(* Schneider Machine Expert - Basic project P1_Part1C, file version 1.6.0.0 *)
(* ProjectInformations: Name=New project *)

HARDWARE
  Cpu 0: TM221M16R/G
  EthernetConfiguration: NetworkName=M221, IpAllocationMode=FixedAddress, IpAddress=0.0.0.0, SubnetMask=0.0.0.0
  SerialLineConfiguration: Baud=Baud19200, Parity=ParityEven, DataBits=DataBits8, StopBits=StopBits1, PhysicalMedium=PhysicalMediumRs485, TransmissionMode=TransmissionModeModbusRtu, SlaveId=1, Addressing=SlaveAddressing
  MastTask: UsePeriodScanMode=false, PeriodScan=100
  FastTask: Period=255, FastTaskSubroutine=On-Off Loop Timer Control
  CpuBehavior: StartingMode=StartAsPreviousState, AutoSaveRamOnEeprom=true, WatchdogPeriod=250

SYMBOLS  (address, symbol, comment, settings)
  %M0       OUTPUT_0_ST
  %M1       START_TIMER_ON
  %M2       DELAY_TIMER_ON
  %MW0      CURRENT_PRESSURE
  %KW0      PRESSURE_CHECKPOINT  [Value=500]
  %KW1      PRESSURE_CHECKPOINT_UNREACHABLE  [Value=1001]
  %TM0      START_TIMER  [Preset=0, Base=OneSecond]
  %TM1      DELAY_TIMER  [Preset=0, Base=OneSecond]
  %I0.0     INPUT_0
  %Q0.0     OUTPUT_0
  %IW0.0    ON_TIMER  [Type=Type_0_10V, Scope=Scope_Normal, Minimum=0, Maximum=1000]
  %IW0.1    OFF_TIMER  [Type=Type_0_10V, Scope=Scope_Normal, Minimum=0, Maximum=1000]

POU I/O Controller
  (* SectionNumber=1 *)

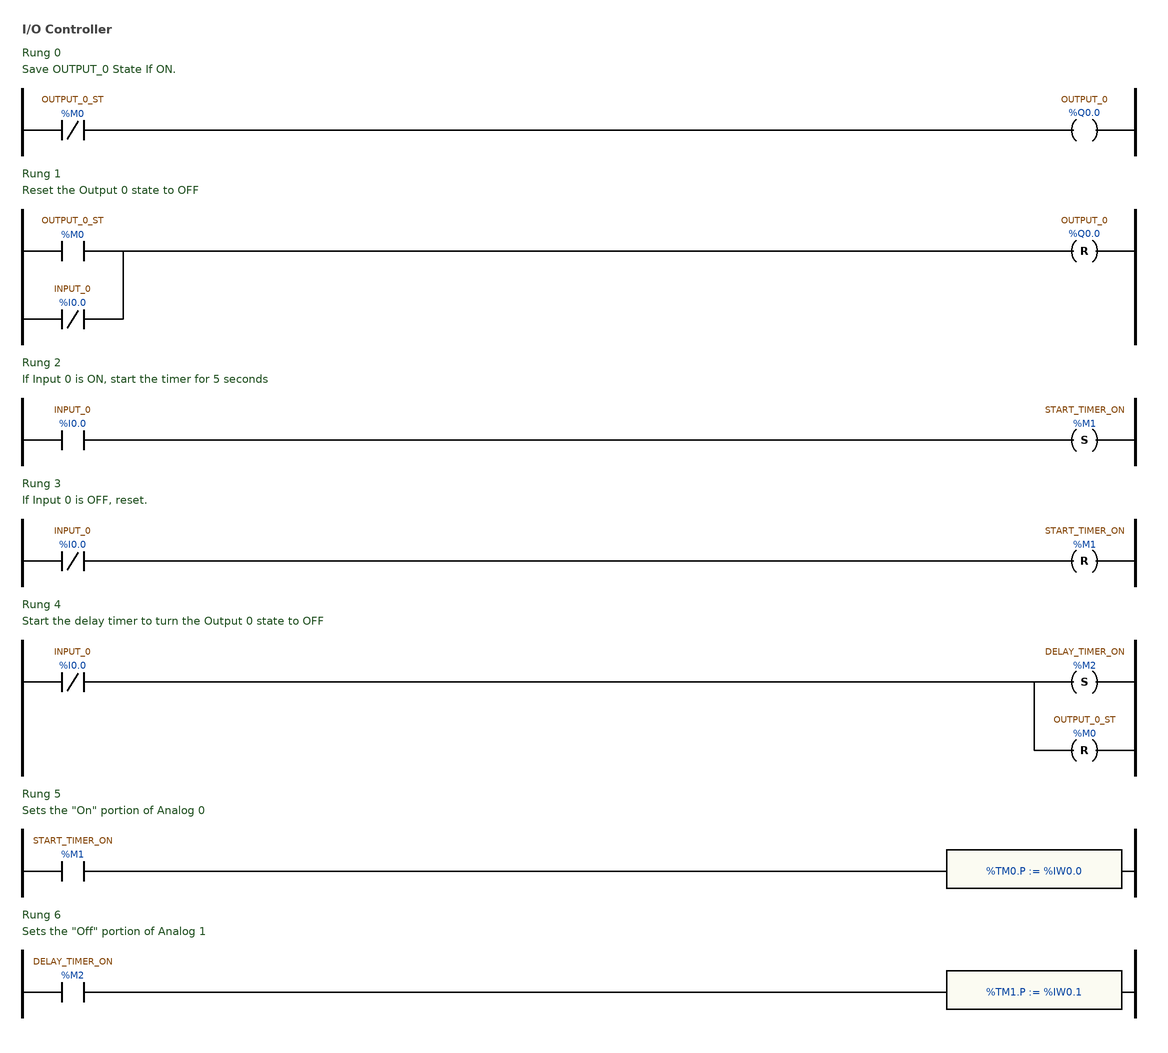

// Rung 0
// Save OUTPUT_0 State If ON.
  LDN %M0                 (* OUTPUT_0_ST *)
  ST %Q0.0                (* OUTPUT_0 *)
  // as ST:
  //   OUTPUT_0 := NOT OUTPUT_0_ST;

// Rung 1
// Reset the Output 0 state to OFF
  LD %M0                  (* OUTPUT_0_ST *)
  ORN %I0.0               (* INPUT_0 *)
  R %Q0.0                 (* OUTPUT_0 *)
  // as ST:
  //   IF OUTPUT_0_ST OR NOT INPUT_0 THEN OUTPUT_0 := FALSE; END_IF;

// Rung 2
// If Input 0 is ON, start the timer for 5 seconds
  LD %I0.0                (* INPUT_0 *)
  S %M1                   (* START_TIMER_ON *)
  // as ST:
  //   IF INPUT_0 THEN START_TIMER_ON := TRUE; END_IF;

// Rung 3
// If Input 0 is OFF, reset.
  LDN %I0.0               (* INPUT_0 *)
  R %M1                   (* START_TIMER_ON *)
  // as ST:
  //   IF NOT INPUT_0 THEN START_TIMER_ON := FALSE; END_IF;

// Rung 4
// Start the delay timer to turn the Output 0 state to OFF
  LDN %I0.0               (* INPUT_0 *)
  S %M2                   (* DELAY_TIMER_ON *)
  R %M0                   (* OUTPUT_0_ST *)
  // as ST:
  //   IF NOT INPUT_0 THEN DELAY_TIMER_ON := TRUE; END_IF;
  //   IF NOT INPUT_0 THEN OUTPUT_0_ST := FALSE; END_IF;

// Rung 5
// Sets the "On" portion of Analog 0
  LD %M1                  (* START_TIMER_ON *)
  [ %TM0.P := %IW0.0 ]    (* START_TIMER, ON_TIMER *)
  // as ST:
  //   IF START_TIMER_ON THEN START_TIMER.P := ON_TIMER; END_IF;

// Rung 6
// Sets the "Off" portion of Analog 1
  LD %M2                  (* DELAY_TIMER_ON *)
  [ %TM1.P := %IW0.1 ]    (* DELAY_TIMER, OFF_TIMER *)
  // as ST:
  //   IF DELAY_TIMER_ON THEN DELAY_TIMER.P := OFF_TIMER; END_IF;

Subroutine On-Off Loop Timer Control
  (* SectionNumber=2, Number=0, IsFastTask=true *)

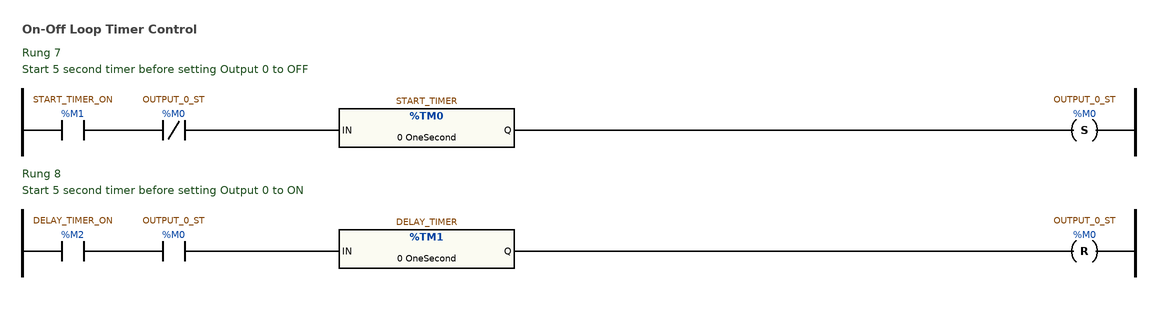

// Rung 7
// Start 5 second timer before setting Output 0 to OFF
  BLK %TM0                (* START_TIMER *)
  LD %M1                  (* START_TIMER_ON *)
  ANDN %M0                (* OUTPUT_0_ST *)
  IN
  OUT_BLK
  LD Q
  S %M0                   (* OUTPUT_0_ST *)
  END_BLK
  // as ST:
  //   START_TIMER(IN := START_TIMER_ON AND NOT OUTPUT_0_ST);
  //   IF START_TIMER.Q THEN OUTPUT_0_ST := TRUE; END_IF;

// Rung 8
// Start 5 second timer before setting Output 0 to ON
  BLK %TM1                (* DELAY_TIMER *)
  LD %M2                  (* DELAY_TIMER_ON *)
  AND %M0                 (* OUTPUT_0_ST *)
  IN
  OUT_BLK
  LD Q
  R %M0                   (* OUTPUT_0_ST *)
  END_BLK
  // as ST:
  //   DELAY_TIMER(IN := DELAY_TIMER_ON AND OUTPUT_0_ST);
  //   IF DELAY_TIMER.Q THEN OUTPUT_0_ST := FALSE; END_IF;
